// Block: BTrk

DATA_BLOCK BTrk
VERSION : 0.1
   NON_RETAIN
   VAR
      Last_B_ID : DInt;
      Empty : BTrk_item;
      EmptyLayer : Array[1..BTRK_LAYER_ITEMS] of BTrk_item;
      EmptyLayers : Struct
         Layer : Array[1..BTRK_LAYER_ITEMS] of BTrk_item;
      END_STRUCT;
      A0301 : Struct
         Empty : Bool;
         MultipleOrders : Bool;
         O_ID : DInt;
         Beam_Qty : Int;
         Beam_Len : Real;
         Beam_W_A : Real;
         Beam_H_B : Real;
         B : Array[1..BTRK_A0301_ITEMS] of BTrk_item;
      END_STRUCT;
      A0302_ENTRY : Struct
         Empty : Bool;
         MultipleOrders : Bool;
         O_ID : DInt;
         Beam_Qty : Int;
         Beam_Len : Real;
         Beam_W_A : Real;
         Beam_H_B : Real;
         B : Array[1..BTRK_A0302_ENTRY_ITEMS] of BTrk_item;
      END_STRUCT;
      A0302_EXIT : Struct
         Empty : Bool;
         MultipleOrders : Bool;
         O_ID : DInt;
         Beam_Qty : Int;
         Beam_Len : Real;
         Beam_W_A : Real;
         Beam_H_B : Real;
         B : Array[1..BTRK_A0302_EXIT_ITEMS] of BTrk_item;
      END_STRUCT;
      A03_EXIT_TOCHECK : Struct
         Empty : Bool;
         Beam_Qty : Int;
         B : Array[1..BTRK_A03_EXIT_TOCHECK_ITEMS] of BTrk_item;
      END_STRUCT;
      A0303 : Struct
         Preparation : Struct
            Empty : Bool;
            Completato : Bool;
            MultipleOrders : Bool;
            O_ID : DInt;
            BeamsPerLayer_Target : Int;
            Layers_Target : Int;
            Beam_Qty : Int;
            Beam_Len : Real;
            Beam_W_A : Real;
            Beam_H_B : Real;
            B : BTrk_item;
            Layer : Array[1..BTRK_LAYER_ITEMS] of BTrk_item;
         END_STRUCT;
         Transfert : Struct
            Empty : Bool;
            MultipleOrders : Bool;
            O_ID : DInt;
            BeamsPerLayer_Target : Int;
            Layers_Target : Int;
            Beams_Qty : Int;
            Beams_Len : Real;
            Beams_W_A : Real;
            Beams_H_B : Real;
            Layer : Array[1..BTRK_LAYER_ITEMS] of BTrk_item;
         END_STRUCT;
         Stacker : Struct
            Empty : Bool;
            Completato : Bool;
            MultipleOrders : Bool;
            O_ID : DInt;
            BeamsPerLayer_Target : Int;
            Layers_Target : Int;
            Layers_Qty : Int;
            Beams_Qty : Int;
            Beams_Len : Real;
            Beams_W_A : Real;
            Beams_H_B : Real;
            Layers : Struct
               Layer : Array[1..BTRK_LAYER_ITEMS] of BTrk_item;
            END_STRUCT;
         END_STRUCT;
      END_STRUCT;
      A0304 : Struct
         Empty : Bool;
         MultipleOrders : Bool;
         NavettaInReggiatura : Bool;
         ReggiaturaConclusa : Bool;
         PaccoRimosso : Bool;
         AbilitazioneCancellazioneDatiPacco : Bool;
         O_ID : DInt;
         BeamsPerLayer_Target : Int;
         Layers_Target : Int;
         Layers_Qty : Int;
         Beams_Qty : Int;
         Beams_Len : Real;
         Beams_W_A : Real;
         Beams_H_B : Real;
         Layers : Struct
            Layer : Array[1..BTRK_LAYER_ITEMS] of BTrk_item;
         END_STRUCT;
      END_STRUCT;
   END_VAR

BEGIN
   // No initialization required
END_DATA_BLOCK
